FUNCTION_BLOCK EcMasterGetDeviceCRC IMPLEMENTS IEcTask
VAR_INPUT
END_VAR
VAR_OUTPUT
END_VAR
VAR
	iState : INT;
	getDeviceCRC : Tc2_EtherCAT.FB_EcGetSlaveCrcErrorEx;
	_execute: BOOL;
	_done: BOOL;
	_busy: BOOL;
	_error: BOOL;
	_netId: AMSNETID;
END_VAR

CASE iState OF
	0:
		IF _execute THEN
			_done := FALSE;
			_busy := TRUE;
			_error := FALSE;
			getDeviceCRC.bExecute := TRUE;
			IF getDeviceCRC.bBusy THEN
				iState := 10;
				_execute := false;
			END_IF
		END_IF
	10:
		IF NOT getDeviceCRC.bBusy THEN
			IF NOT getDeviceCRC.bError THEN
				_done := TRUE;
			ELSE
				_error := TRUE;
			END_IF
			_busy := FALSE;
			getDeviceCRC.bExecute := FALSE;
			iState := 0;
		END_IF
END_CASE

getDeviceCRC(sNetId := Tc2_System.F_CreateAmsNetId(nIds := NetId));

{warning 'add method implementation '}
METHOD Abort : BOOL
getDeviceCRC.bExecute := FALSE;
_busy := FALSE;
_execute := FALSE;
Abort := TRUE;
iState := 0;
END_METHOD

{warning 'add property implementation'}
PROPERTY Busy : BOOL
GET
Busy := _busy;
END_GET
END_PROPERTY

PROPERTY DeviceAddr : uint
GET
DeviceAddr := getDeviceCRC.nSlaveAddr;
END_GET
SET
getDeviceCRC.nSlaveAddr := DeviceAddr;
END_SET
END_PROPERTY

PROPERTY DeviceCRC :  ST_EcCrcErrorEx
GET
DeviceCRC := getDeviceCRC.crcError;
END_GET
END_PROPERTY

{warning 'add property implementation'}
PROPERTY Done : BOOL
GET
Done := _done;
END_GET
END_PROPERTY

{warning 'add property implementation'}
PROPERTY Error : BOOL
GET
Error := _error;
END_GET
END_PROPERTY

{warning 'add method implementation '}
METHOD Execute : BOOL
IF NOT getDeviceCRC.bBusy THEN
	Execute := _execute := true;
END_IF
END_METHOD

{warning 'add property implementation'}
PROPERTY NetID : amsnetid
GET
NetID := _netId;
END_GET
SET
_netId := NetID;
END_SET
END_PROPERTY

END_FUNCTION_BLOCK

(* stored: Version 1.1.0.1, ProductVersion 3.1.4024.9
   POU EcMasterGetDeviceCRC: Id {b134bf75-2d16-450b-90bf-d567390a3f26}, SpecialFunc None
   Method Abort: Id {9233e0e0-5278-4efe-b24b-b972bfa1f7df}
   Property Busy: Id {f4f81a6d-8453-4613-877f-6f383dc14282}
   Get Get: Id {4233078c-28d4-48dd-80b0-9e9ae2e15532}
   Property DeviceAddr: Id {7c2aaa9b-1551-4a8c-81d9-fe8515b143db}
   Get Get: Id {70a7ca5b-63de-4420-ba5d-759552805a5c}
   Set Set: Id {ecdd739f-4c51-4243-98e8-6a86c5ec1c29}
   Property DeviceCRC: Id {ee643b98-b9dd-4aa2-b240-e4e420bed4ed}
   Get Get: Id {e0288b1e-8e63-45a1-af06-cb7b43d00170}
   Property Done: Id {b2f7288b-191f-4b92-91fa-4a75f1639168}
   Get Get: Id {d42635a3-eacc-40cf-8218-ec4a5e53bb76}
   Property Error: Id {f7351aba-5c87-4091-a30d-c6b267ffefef}
   Get Get: Id {d9ab0c8b-d959-427a-ade3-227f59981d06}
   Method Execute: Id {0ca5408f-4c0d-48ef-be70-2414b2d2a7e3}
   Property NetID: Id {f7479886-ad80-40ff-a160-c2333a320f11}
   Get Get: Id {0883fade-120f-48ea-85ea-b6e101953aeb}
   Set Set: Id {186eb6ca-1018-4ce0-b385-460ff4c05f06} *)
